PROGRAM MAIN
VAR
	EventBuffer : FB_EventBuffer;
	
	AddEvent : BOOL;
	stEventAdd : ST_Event;
	bErrorToAddEvent : BOOL;
	
	ReadAndRemoveEvent : BOOL;
	LastReadEvent : ST_Event;
	bErrorToReadRemoveEvent : BOOL;
	
END_VAR

IF AddEvent THEN
	EventBuffer.AddEvent(stEvent := stEventAdd, bError => bErrorToAddEvent);
	AddEvent := FALSE;
END_IF
IF ReadAndRemoveEvent THEN
	EventBuffer.GetRemoveEvent(stEvent => LastReadEvent, bError => bErrorToReadRemoveEvent);
	ReadAndRemoveEvent := FALSE;
END_IF

END_PROGRAM

(* stored: Version 1.1.0.1, ProductVersion 3.1.4024.12
   POU MAIN: Id {763b6711-ecff-46da-8c71-1268c29893eb}, SpecialFunc None *)
